FUNCTION_BLOCK FB_AX5000 EXTENDS FB_AxisNc
VAR_INPUT
END_VAR
VAR_OUTPUT
END_VAR
VAR_IN_OUT
	stDriveRef 			: ST_DRIVEREF;
END_VAR
VAR
	//variables for the hardware reset 
	fbTrigNotBusy		: F_TRIG;
	bNotBusy			: BOOL;
	fbTrigResetNotBusy	: F_TRIG;
	fbSOEReset			: FB_SoEReset;
END_VAR

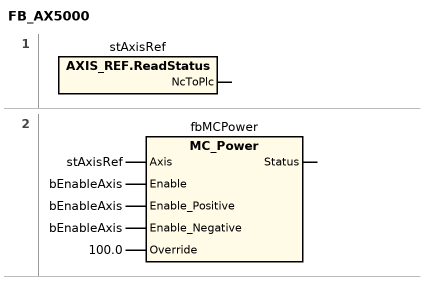
// NETWORK 1
stAxisRef.ReadStatus();

// NETWORK 2
//   fbMCPower: Enable
fbMCPower(
    Axis := stAxisRef,
    Enable := bEnableAxis,
    Enable_Positive := bEnableAxis,
    Enable_Negative := bEnableAxis,
    Override := 100.0); // MC_Power

METHOD PUBLIC M_HardwareReset : UDINT
//This method override the hardware reset method of the Inherited FB_AxisBlock
//in order to perform commands specific to resetting an AX5000 Drive
VAR_INPUT
	bReset : BOOL;
END_VAR
//Result of the Reset method is 
// 0 : Idle
// 1 : busy
// 3 : complete
// > 3 Error returned by associated function blocks
VAR
	
	
END_VAR
VAR_INST // added by the converter: edge detectors and wires of the graphical bodies
    _w1, _w2 : BOOL;
END_VAR
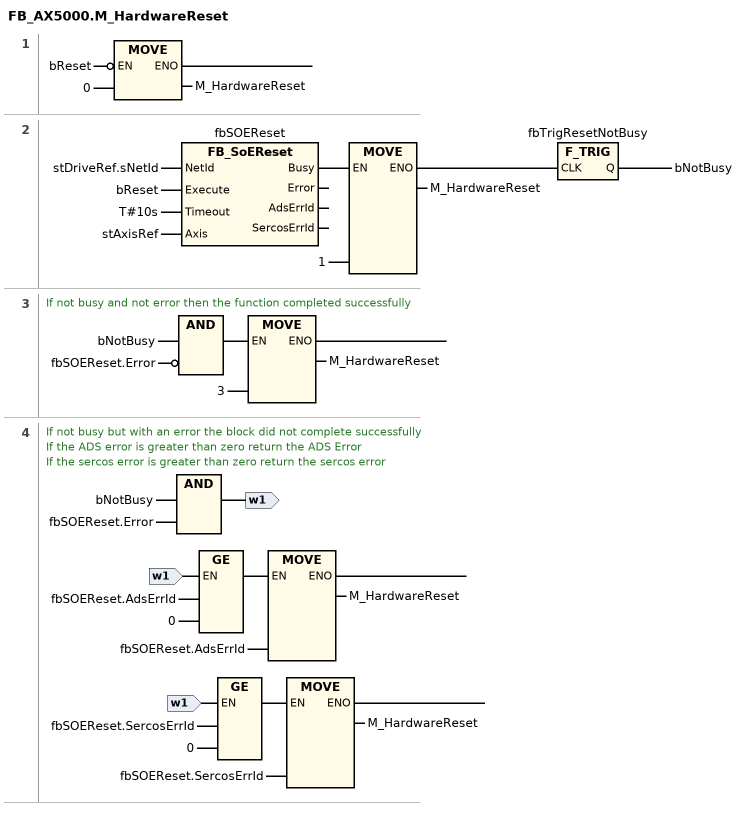
// NETWORK 1
IF NOT bReset THEN M_HardwareReset := 0; END_IF

// NETWORK 2
fbSOEReset(NetId := stDriveRef.sNetId, Execute := bReset, Timeout := T#10s, Axis := stAxisRef); // FB_SoEReset
_w1 := fbSOEReset.Busy;
IF _w1 THEN M_HardwareReset := 1; END_IF
fbTrigResetNotBusy(CLK := _w1); // F_TRIG
bNotBusy := fbTrigResetNotBusy.Q;

// NETWORK 3
// If not busy and not error then the function completed successfully
IF bNotBusy AND NOT fbSOEReset.Error THEN M_HardwareReset := 3; END_IF

// NETWORK 4
// If not busy but with an error the block did not complete successfully
// If the ADS error is greater than zero return the ADS Error
// If the sercos error is greater than zero return the sercos error
_w2 := bNotBusy AND fbSOEReset.Error;
IF _w2 AND fbSOEReset.AdsErrId >= 0 THEN M_HardwareReset := fbSOEReset.AdsErrId; END_IF
IF _w2 AND fbSOEReset.SercosErrId >= 0 THEN M_HardwareReset := fbSOEReset.SercosErrId; END_IF
END_METHOD

END_FUNCTION_BLOCK

(* stored: Version 1.1.0.1, ProductVersion 3.1.4024.11
   POU FB_AX5000: Id {84154bdf-9edb-4eb2-ba69-2536319b1bd8}, SpecialFunc None
   Method M_HardwareReset: Id {54909ba6-d11d-4f71-b639-8ed98c6eb9e3} *)
